Fanuc TP program (LS listing): METALWIT.LS

/PROG  METALWIT	  Collection
/ATTR
OWNER		= MNEDITOR;
COMMENT		= "";
PROG_SIZE	= 1594;
CREATE		= DATE 25-05-14  TIME 13:33:34;
MODIFIED	= DATE 26-04-29  TIME 10:40:50;
FILE_NAME	= ;
VERSION		= 0;
LINE_COUNT	= 63;
MEMORY_SIZE	= 2346;
PROTECT		= READ_WRITE;
TCD:  STACK_SIZE	= 0,
      TASK_PRIORITY	= 50,
      TIME_SLICE	= 0,
      BUSY_LAMP_OFF	= 0,
      ABORT_REQUEST	= 0,
      PAUSE_REQUEST	= 0;
DEFAULT_GROUP	= *,*,*,*,*;
CONTROL_CODE	= 00000000 00000000;
/MN
   1:  CALL BLOW_CIRCLE    ;
   2:  CALL GO_TABLE_T1    ;
   3:  CALL GO_TABLE_T2    ;
   4:  CALL GO_HOME_TABLE_T2    ;
   5:  CALL GO_HOME_TABLE_T1    ;
   6:  CALL MODE_3    ;
   7:  CALL DOOR_NOT_OP    ;
   8:  CALL DOOR_OP_COND    ;
   9:  CALL BASE_MOVED    ;
  10:  CALL BASE_RDY_COND    ;
  11:  CALL START_CNC    ;
  12:  CALL CROSS_CONNECTION    ;
  13:  CALL DROP_T2    ;
  14:  CALL PICK_UP_T2    ;
  15:  CALL DROP_T1    ;
  16:  CALL PICK_UP_T1    ;
  17:  CALL STOP_BLOW    ;
  18:  CALL START_BLOW    ;
  19:  CALL DOOR_COND    ;
  20:  CALL DOOR_ERR    ;
  21:  CALL PICK_TRAY_T2    ;
  22:  CALL T1_DET_LOST    ;
  23:  CALL T1_GRIP_COND    ;
  24:  CALL T2_DET_LOST    ;
  25:  CALL T2_GRIP_COND    ;
  26:  CALL CLOSE_T2    ;
  27:  CALL CLOSE_T1    ;
  28:  CALL OPEN_T2    ;
  29:  CALL OPEN_T1    ;
  30:  CALL MODE_2    ;
  31:  CALL PICK_VICE2_T1    ;
  32:  CALL PICK_VICE2_T2    ;
  33:  CALL PLACE_VICE2_T1    ;
  34:  CALL PLACE_VICE2_T2    ;
  35:  CALL PLACE_VICE1_T2    ;
  36:  CALL PLACE_VICE1_T1    ;
  37:  CALL PICK_VICE1_T2    ;
  38:  CALL PICK_VICE1_T1    ;
  39:  CALL GO_HOME    ;
  40:  CALL GO_TABLE_VICE_T1    ;
  41:  CALL GO_VICE_TABLE_T1    ;
  42:  CALL GO_VICE_TABLE_T2    ;
  43:  CALL CALCULATE_T2    ;
  44:  CALL CALCULATE_T1    ;
  45:  CALL PICK_TRAY_T1    ;
  46:  CALL PLACE_TRAY_T2    ;
  47:  CALL PLACE_TRAY_T1    ;
  48:  CALL PICK_TRAY_1    ;
  49:  CALL GO_TABLE_VICE_T2    ;
  50:  CALL MODE_1    ;
  51:  CALL SET_SPC    ;
  52:  CALL CLOSE_DOOR    ;
  53:  CALL OPEN_DOOR    ;
  54:  CALL GO_TABLE_VICE    ;
  55:  CALL TEST    ;
  56:  CALL PLACE_VICE1    ;
  57:  CALL PLACE_TRAY    ;
  58:  CALL PICK_VICE1    ;
  59:  CALL PICK_TRAY    ;
  60:  CALL CALCULATE    ;
  61:  CALL ADJ_PR_R    ;
  62:  CALL INITIALIZE    ;
  63:  CALL MAIN    ;
/POS
/END
